(* IEC 61131-3 sources: AXOpen/src/components.kuka.robotics/app/SystemConstants, 3 files *)

(* ---- plc_line_HwIdentifiers.st ---- *)
CONFIGURATION HardwareIDs
    VAR_GLOBAL CONSTANT
        KRC4_HwID : UINT := UINT#258;
        KRC4_DIO512_512_digital_in__and_outputs_HwID : UINT := UINT#262;
        KRC4_KRC4_HwID : UINT := UINT#261;
        KRC4_KRC4_KRC4_ProfiNet_5_0_HwID : UINT := UINT#263;
        KRC4_KRC4_profinet_HwID : UINT := UINT#257;
        KRC4_KRC4_profinet_Port_1_HwID : UINT := UINT#259;
        KRC4_Rack_HwID : UINT := UINT#260;
        plc_line_HwID : UINT := UINT#32;
        plc_line_Rail_0_HwID : UINT := UINT#273;
        plc_line_plc_line_HwID : UINT := UINT#48;
        plc_line_plc_line_CPU_display_1_HwID : UINT := UINT#54;
        plc_line_plc_line_Card_reader_writer_1_HwID : UINT := UINT#51;
        plc_line_plc_line_DP_interface_1_HwID : UINT := UINT#60;
        plc_line_plc_line_OPC_UA_1_HwID : UINT := UINT#117;
        plc_line_plc_line_Virtual_communication_interface_HwID : UINT := UINT#135;
        plc_line_plc_line_profinet_x1_HwID : UINT := UINT#64;
        plc_line_plc_line_profinet_x1_Port_1_HwID : UINT := UINT#65;
        plc_line_plc_line_profinet_x1_Port_2_HwID : UINT := UINT#66;
        plc_line_plc_line_profinet_x2_HwID : UINT := UINT#72;
        plc_line_plc_line_profinet_x2_Port_3_HwID : UINT := UINT#73;
        profinet_plc_line_HwID : UINT := UINT#256;

    END_VAR
END_CONFIGURATION

(* ---- plc_line_IoAddresses.st ---- *)
CONFIGURATION IoAddresses
    VAR_GLOBAL
        KRC4_DIO512_InputAddress_0 AT %IL0: LWORD;
        KRC4_DIO512_InputAddress_1 AT %IL8: LWORD;
        KRC4_DIO512_InputAddress_2 AT %IL16: LWORD;
        KRC4_DIO512_InputAddress_3 AT %IL24: LWORD;
        KRC4_DIO512_InputAddress_4 AT %IL32: LWORD;
        KRC4_DIO512_InputAddress_5 AT %IL40: LWORD;
        KRC4_DIO512_InputAddress_6 AT %IL48: LWORD;
        KRC4_DIO512_InputAddress_7 AT %IL56: LWORD;
        KRC4_DIO512_OutputAddress_0 AT %QL0: LWORD;
        KRC4_DIO512_OutputAddress_1 AT %QL8: LWORD;
        KRC4_DIO512_OutputAddress_2 AT %QL16: LWORD;
        KRC4_DIO512_OutputAddress_3 AT %QL24: LWORD;
        KRC4_DIO512_OutputAddress_4 AT %QL32: LWORD;
        KRC4_DIO512_OutputAddress_5 AT %QL40: LWORD;
        KRC4_DIO512_OutputAddress_6 AT %QL48: LWORD;
        KRC4_DIO512_OutputAddress_7 AT %QL56: LWORD;

    END_VAR
END_CONFIGURATION

(* ---- plc_main_HwIdentifiers.st ---- *)
CONFIGURATION HardwareIDs
    VAR_GLOBAL CONSTANT
        kuka_rb1_HwID : UINT := UINT#258;
        kuka_rb1_DIO512_512_digital_in__and_outputs_HwID : UINT := UINT#262;
        kuka_rb1_Rack_HwID : UINT := UINT#260;
        kuka_rb1_kuka_rb1_HwID : UINT := UINT#261;
        kuka_rb1_kuka_rb1_Interface1_HwID : UINT := UINT#257;
        kuka_rb1_kuka_rb1_Interface1_Port_1_HwID : UINT := UINT#259;
        kuka_rb1_kuka_rb1_KRC4_ProfiNet_5_0_HwID : UINT := UINT#263;
        plc_main_HwID : UINT := UINT#32;
        plc_main_Rail_0_HwID : UINT := UINT#264;
        plc_main_plc_main_HwID : UINT := UINT#48;
        plc_main_plc_main_CPU_display_1_HwID : UINT := UINT#54;
        plc_main_plc_main_Card_reader_writer_1_HwID : UINT := UINT#51;
        plc_main_plc_main_OPC_UA_1_HwID : UINT := UINT#117;
        plc_main_plc_main_PROFINET_interface_1_HwID : UINT := UINT#64;
        plc_main_plc_main_PROFINET_interface_1_Port_1_HwID : UINT := UINT#65;
        plc_main_plc_main_PROFINET_interface_1_Port_2_HwID : UINT := UINT#66;
        plc_main_plc_main_PROFINET_interface_2_HwID : UINT := UINT#72;
        plc_main_plc_main_PROFINET_interface_2_Port_3_HwID : UINT := UINT#73;
        plc_main_plc_main_PROFINET_interface_2_Port_4_HwID : UINT := UINT#74;
        plc_main_plc_main_PROFINET_interface_GBIT_3_HwID : UINT := UINT#120;
        plc_main_plc_main_PROFINET_interface_GBIT_3_Port_5_HwID : UINT := UINT#121;
        plc_main_plc_main_Virtual_communication_interface_HwID : UINT := UINT#135;
        profinet_plc_main_HwID : UINT := UINT#256;

    END_VAR
END_CONFIGURATION
